PROGRAM prgRWLynus
VAR
	fbRW1		: FB_ReadWrite_V2;
END_VAR



fbRW1(
	eUploadType:= 2 , 
	bBusy=> , 
	bError=> , 
	udiErrorCodeOut=> , 
	eErrorReadWrite_Out=> );

END_PROGRAM

(* stored: Version 1.1.0.1, ProductVersion 3.1.4024.11
   POU prgRWLynus: Id {aff76794-a195-49b5-a617-4aeaae11f21d}, SpecialFunc None *)
